PROGRAM updateMotors
VAR
END_VAR

GVL_devices.fbLftWidthMotor();
GVL_devices.fbRhtWidthMotor();

GVL_devices.fbLftClampMotor();
GVL_devices.fbRhtClampMotor();

GVL_devices.fbLftRotationMotor();	
GVL_devices.fbRhtRotationMotor();	

GVL_devices.fbColumn0Motor();	
GVL_devices.fbColumn1Motor();	
GVL_devices.fbColumn2Motor();	
GVL_devices.fbColumn3Motor();

END_PROGRAM

(* stored: Version 1.1.0.1, ProductVersion 3.1.4024.13
   POU updateMotors: Id {113379e0-5e5f-48bf-b344-8890dfe42f80}, SpecialFunc None *)
